SYSTEM ShiftForkCaseStudy
  (* Version 1.0, 2022-12-15, AK124017 *)
  APPLICATION ShiftForkCaseStudyApp
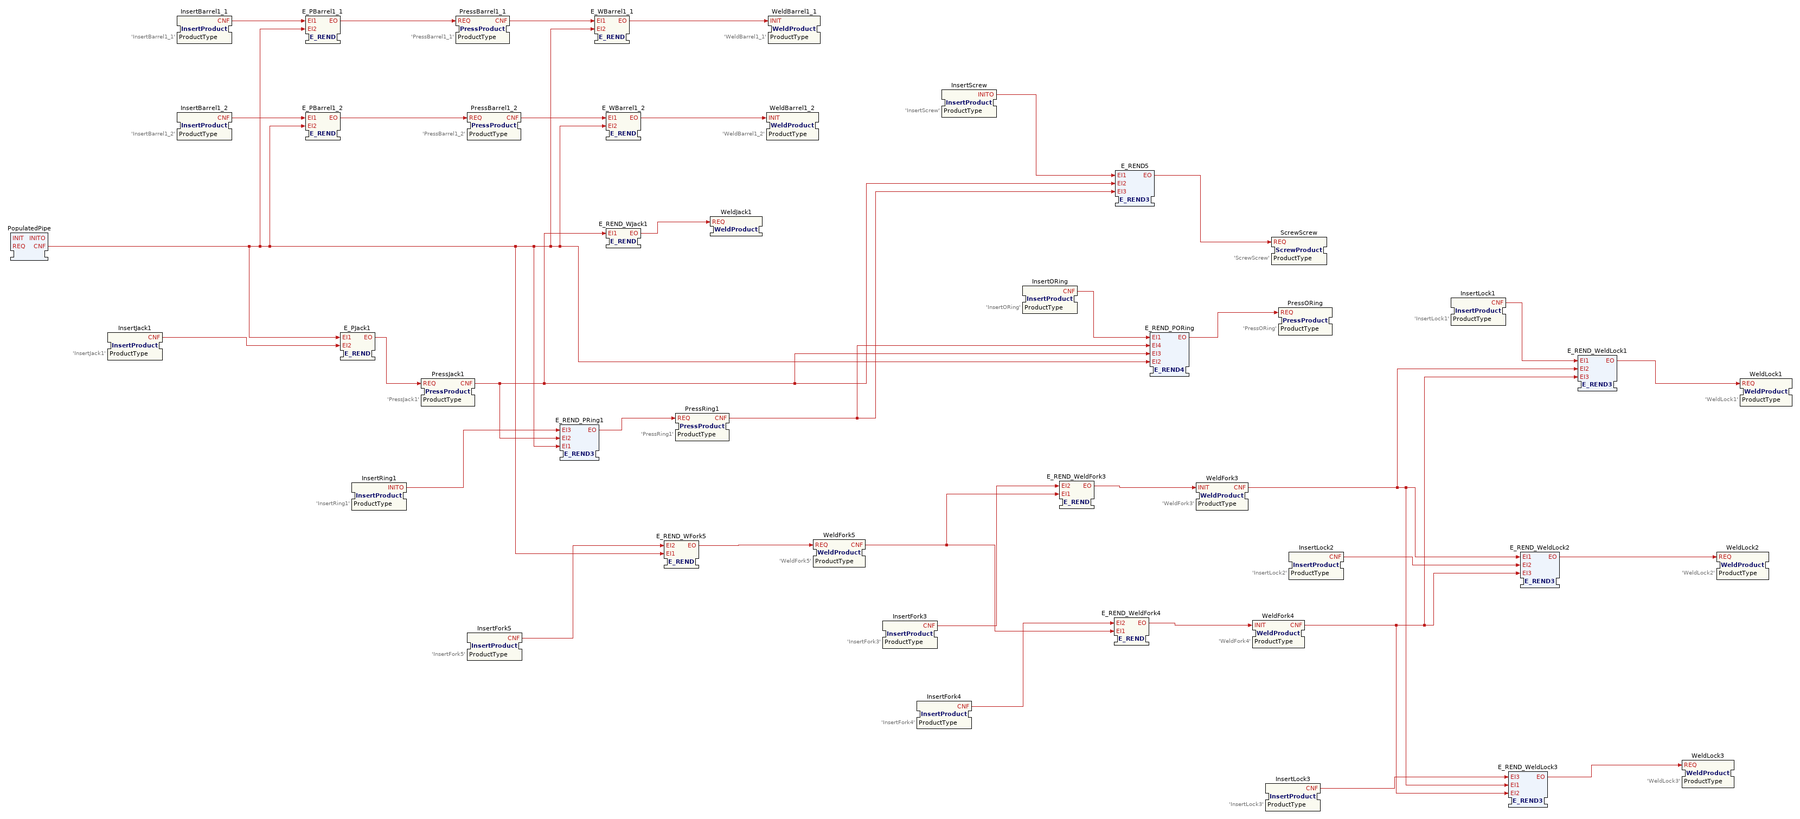
    FBS
      InsertFork5 : InsertProduct(ProductType := 'InsertFork5');
      WeldFork5 : WeldProduct(ProductType := 'WeldFork5');
      InsertFork3 : InsertProduct(ProductType := 'InsertFork3');
      WeldFork3 : WeldProduct(ProductType := 'WeldFork3');
      InsertFork4 : InsertProduct(ProductType := 'InsertFork4');
      WeldFork4 : WeldProduct(ProductType := 'WeldFork4');
      InsertLock1 : InsertProduct(ProductType := 'InsertLock1');
      InsertLock2 : InsertProduct(ProductType := 'InsertLock2');
      InsertLock3 : InsertProduct(ProductType := 'InsertLock3');
      WeldLock1 : WeldProduct(ProductType := 'WeldLock1');
      WeldLock2 : WeldProduct(ProductType := 'WeldLock2');
      WeldLock3 : WeldProduct(ProductType := 'WeldLock3');
      E_REND_WeldFork3 : E_REND;
      E_REND_WeldFork4 : E_REND;
      PressRing1 : PressProduct(ProductType := 'PressRing1');
      InsertORing : InsertProduct(ProductType := 'InsertORing');
      InsertJack1 : InsertProduct(ProductType := 'InsertJack1');
      PressJack1 : PressProduct(ProductType := 'PressJack1');
      InsertScrew : InsertProduct(ProductType := 'InsertScrew');
      InsertRing1 : InsertProduct(ProductType := 'InsertRing1');
      ScrewScrew : ScrewProduct(ProductType := 'ScrewScrew');
      PressORing : PressProduct(ProductType := 'PressORing');
      PressBarrel1_1 : PressProduct(ProductType := 'PressBarrel1_1');
      InsertBarrel1_1 : InsertProduct(ProductType := 'InsertBarrel1_1');
      WeldBarrel1_1 : WeldProduct(ProductType := 'WeldBarrel1_1');
      PressBarrel1_2 : PressProduct(ProductType := 'PressBarrel1_2');
      WeldBarrel1_2 : WeldProduct(ProductType := 'WeldBarrel1_2');
      InsertBarrel1_2 : InsertProduct(ProductType := 'InsertBarrel1_2');
      WeldJack1 : WeldProduct;
      E_WBarrel1_1 : E_REND;
      E_WBarrel1_2 : E_REND;
      E_REND_WJack1 : E_REND;
      E_REND_WFork5 : E_REND;
      E_PBarrel1_1 : E_REND;
      E_PBarrel1_2 : E_REND;
      E_PJack1 : E_REND;
    END_FBS
    SUBAPPS
      E_REND_PRing1 : E_REND3;
      E_REND_PORing : E_REND4;
      E_REND5 : E_REND3;
      E_REND_WeldLock1 : E_REND3;
      E_REND_WeldLock2 : E_REND3;
      E_REND_WeldLock3 : E_REND3;
    END_SUBAPPS
    SUBAPPLICATION PopulatedPipe
      EVENT_INPUT
        INIT;
        REQ;
      END_EVENT
      EVENT_OUTPUT
        INITO;
        CNF;
      END_EVENT
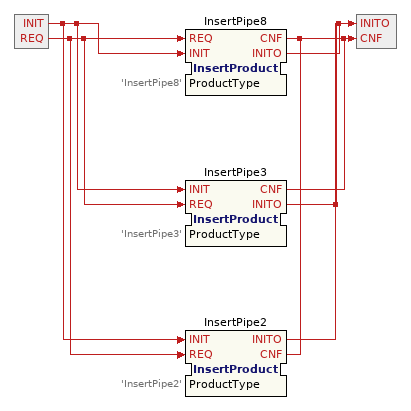
      FBS
        InsertPipe2 : InsertProduct(ProductType := 'InsertPipe2');
        InsertPipe3 : InsertProduct(ProductType := 'InsertPipe3');
        InsertPipe8 : InsertProduct(ProductType := 'InsertPipe8');
      END_FBS
      EVENT_CONNECTIONS
        INIT TO InsertPipe2.INIT;
        REQ TO InsertPipe2.REQ;
        INIT TO InsertPipe3.INIT;
        REQ TO InsertPipe3.REQ;
        REQ TO InsertPipe8.REQ;
        INIT TO InsertPipe8.INIT;
        InsertPipe2.INITO TO INITO;
        InsertPipe2.CNF TO CNF;
        InsertPipe3.CNF TO CNF;
        InsertPipe3.INITO TO INITO;
        InsertPipe8.CNF TO CNF;
        InsertPipe8.INITO TO INITO;
      END_CONNECTIONS
    END_SUBAPPLICATION
    EVENT_CONNECTIONS
      InsertFork3.CNF TO E_REND_WeldFork3.EI2;
      WeldFork5.CNF TO E_REND_WeldFork3.EI1;
      E_REND_WeldFork3.EO TO WeldFork3.INIT;
      InsertFork4.CNF TO E_REND_WeldFork4.EI2;
      WeldFork5.CNF TO E_REND_WeldFork4.EI1;
      E_REND_WeldFork4.EO TO WeldFork4.INIT;
      PressBarrel1_1.CNF TO E_WBarrel1_1.EI1;
      E_WBarrel1_1.EO TO WeldBarrel1_1.INIT;
      PressBarrel1_2.CNF TO E_WBarrel1_2.EI1;
      E_WBarrel1_2.EO TO WeldBarrel1_2.INIT;
      PressJack1.CNF TO E_REND_WJack1.EI1;
      E_REND_WJack1.EO TO WeldJack1.REQ;
      E_REND_PRing1.EO TO PressRing1.REQ;
      InsertORing.CNF TO E_REND_PORing.EI1;
      E_REND_PORing.EO TO PressORing.REQ;
      InsertScrew.INITO TO E_REND5.EI1;
      PressJack1.CNF TO E_REND5.EI2;
      PressRing1.CNF TO E_REND5.EI3;
      E_REND5.EO TO ScrewScrew.REQ;
      E_REND_WFork5.EO TO WeldFork5.REQ;
      InsertLock1.CNF TO E_REND_WeldLock1.EI1;
      E_REND_WeldLock1.EO TO WeldLock1.REQ;
      WeldFork3.CNF TO E_REND_WeldLock1.EI2;
      WeldFork4.CNF TO E_REND_WeldLock1.EI3;
      WeldFork3.CNF TO E_REND_WeldLock2.EI1;
      InsertLock2.CNF TO E_REND_WeldLock2.EI2;
      WeldFork4.CNF TO E_REND_WeldLock2.EI3;
      E_REND_WeldLock2.EO TO WeldLock2.REQ;
      InsertLock3.CNF TO E_REND_WeldLock3.EI3;
      WeldFork3.CNF TO E_REND_WeldLock3.EI1;
      WeldFork4.CNF TO E_REND_WeldLock3.EI2;
      E_REND_WeldLock3.EO TO WeldLock3.REQ;
      E_PBarrel1_1.EO TO PressBarrel1_1.REQ;
      InsertBarrel1_1.CNF TO E_PBarrel1_1.EI1;
      InsertBarrel1_2.CNF TO E_PBarrel1_2.EI1;
      E_PBarrel1_2.EO TO PressBarrel1_2.REQ;
      PopulatedPipe.CNF TO E_PBarrel1_1.EI2;
      PopulatedPipe.CNF TO E_WBarrel1_1.EI2;
      PopulatedPipe.CNF TO E_PBarrel1_2.EI2;
      PopulatedPipe.CNF TO E_WBarrel1_2.EI2;
      E_PJack1.EO TO PressJack1.REQ;
      PopulatedPipe.CNF TO E_PJack1.EI1;
      InsertJack1.CNF TO E_PJack1.EI2;
      InsertRing1.INITO TO E_REND_PRing1.EI3;
      PressJack1.CNF TO E_REND_PRing1.EI2;
      PopulatedPipe.CNF TO E_REND_PRing1.EI1;
      PressRing1.CNF TO E_REND_PORing.EI4;
      PressJack1.CNF TO E_REND_PORing.EI3;
      PopulatedPipe.CNF TO E_REND_PORing.EI2;
      InsertFork5.CNF TO E_REND_WFork5.EI2;
      PopulatedPipe.CNF TO E_REND_WFork5.EI1;
    END_CONNECTIONS
  END_APPLICATION
END_SYSTEM
